// TIA Portal V16 export
// export: Created 2021-09-08T12:46:05.9952006Z, ExportSetting WithDefaults, DisplayName Totally Integrated Automation Portal, DisplayVersion V16 Update 3, DisplayName TIA Portal Version Control Interface, DisplayVersion V16 Update 2, DisplayName TIA Portal Openness, DisplayVersion V16 Update 3, DisplayName TIA Portal Teamcenter Gateway, DisplayVersion V16, DisplayName STEP 7 Professional, DisplayVersion V16 Update 3, DisplayName STEP 7 Safety, DisplayVersion V16, DisplayName WinCC Advanced, DisplayVersion V16 Update 3
ORGANIZATION_BLOCK "Main"   // OB1, LAD, ProgramCycle
TITLE = "Main Program Sweep (Cycle)"
{ S7_Optimized_Access := 'TRUE' }
VERSION : 0.1
// stored: AutoNumber true, IsIECCheckEnabled false, SetENOAutomatically false
   VAR_INPUT
      Initial_Call : Bool;   // Initial call of this OB
      Remanence : Bool;   // =True, if remanent data are available
   END_VAR
BEGIN

REGION Network 1: Клапаны
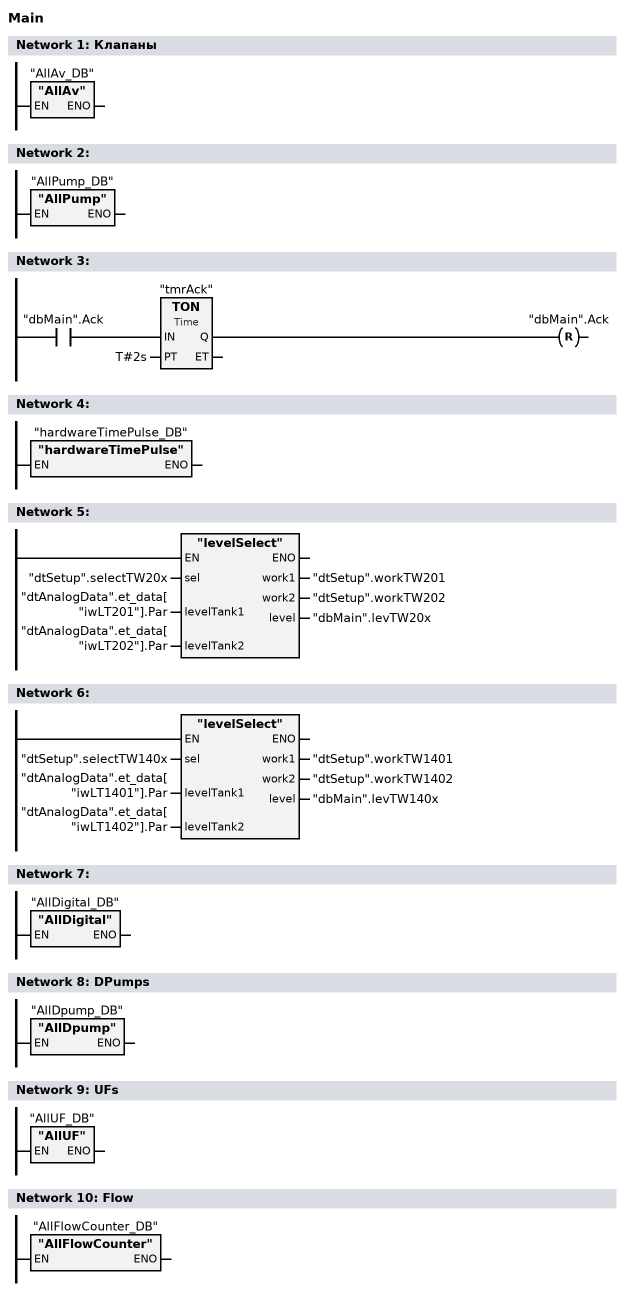
   RUNG wire#powerrail
      "AllAv_DB"()
   END_RUNG
   // the same network as SCL:
   "AllAv_DB"();   // "AllAv"
END_REGION

REGION Network 2
   RUNG wire#powerrail
      "AllPump_DB"()
   END_RUNG
   // the same network as SCL:
   "AllPump_DB"();   // "AllPump"
END_REGION

REGION Network 3
   RUNG wire#powerrail
      Contact( "dbMain".Ack )
      { S7_Templates := "time_type := Time" } "tmrAck".TON(pt := T#2s, et =>)
      R_Coil( "dbMain".Ack )
   END_RUNG
   // the same network as SCL:
   "tmrAck".TON(IN := "dbMain".Ack, PT := T#2s);
   IF "tmrAck".Q THEN "dbMain".Ack := FALSE; END_IF;
END_REGION

REGION Network 4
   RUNG wire#powerrail
      "hardwareTimePulse_DB"()
   END_RUNG
   // the same network as SCL:
   "hardwareTimePulse_DB"();   // "hardwareTimePulse"
END_REGION

REGION Network 5
   RUNG wire#powerrail
      "levelSelect"(sel := "dtSetup".selectTW20x, levelTank1 := "dtAnalogData".et_data["iwLT201"].Par, levelTank2 := "dtAnalogData".et_data["iwLT202"].Par, work1 => "dtSetup".workTW201, work2 => "dtSetup".workTW202, level => "dbMain".levTW20x)
   END_RUNG
   // the same network as SCL:
   "levelSelect"(sel := "dtSetup".selectTW20x,
                 levelTank1 := "dtAnalogData".et_data["iwLT201"].Par,
                 levelTank2 := "dtAnalogData".et_data["iwLT202"].Par,
                 work1 => "dtSetup".workTW201,
                 work2 => "dtSetup".workTW202,
                 level => "dbMain".levTW20x);
END_REGION

REGION Network 6
   RUNG wire#powerrail
      "levelSelect"(sel := "dtSetup".selectTW140x, levelTank1 := "dtAnalogData".et_data["iwLT1401"].Par, levelTank2 := "dtAnalogData".et_data["iwLT1402"].Par, work1 => "dtSetup".workTW1401, work2 => "dtSetup".workTW1402, level => "dbMain".levTW140x)
   END_RUNG
   // the same network as SCL:
   "levelSelect"(sel := "dtSetup".selectTW140x,
                 levelTank1 := "dtAnalogData".et_data["iwLT1401"].Par,
                 levelTank2 := "dtAnalogData".et_data["iwLT1402"].Par,
                 work1 => "dtSetup".workTW1401,
                 work2 => "dtSetup".workTW1402,
                 level => "dbMain".levTW140x);
END_REGION

REGION Network 7
   RUNG wire#powerrail
      "AllDigital_DB"()
   END_RUNG
   // the same network as SCL:
   "AllDigital_DB"();   // "AllDigital"
END_REGION

REGION Network 8: DPumps
   RUNG wire#powerrail
      "AllDpump_DB"()
   END_RUNG
   // the same network as SCL:
   "AllDpump_DB"();   // "AllDpump"
END_REGION

REGION Network 9: UFs
   RUNG wire#powerrail
      "AllUF_DB"()
   END_RUNG
   // the same network as SCL:
   "AllUF_DB"();   // "AllUF"
END_REGION

REGION Network 10: Flow
   RUNG wire#powerrail
      "AllFlowCounter_DB"()
   END_RUNG
   // the same network as SCL:
   "AllFlowCounter_DB"();   // "AllFlowCounter"
END_REGION
END_ORGANIZATION_BLOCK
